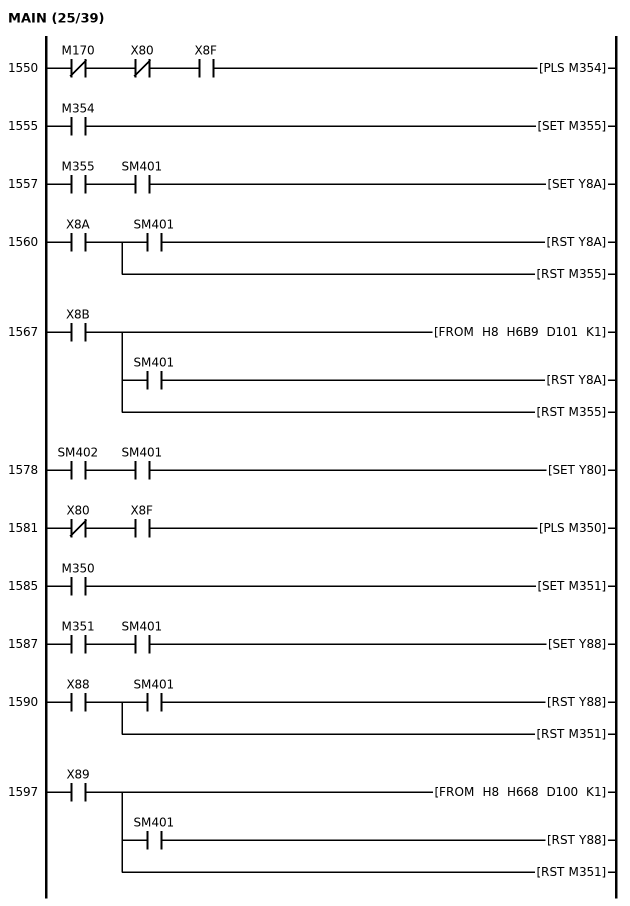
[picture p24: ladder of MAIN, rungs at steps 1550 to 1597]
1550  LDI     M170
      ANI     X80
      AND     X8F
      PLS     M354
1555  LD      M354
      SET     M355
1557  LD      M355
      AND     SM401
      SET     Y8A
1560  LD      X8A
      MPS
      AND     SM401
      RST     Y8A
      MPP
      RST     M355
; 
1567  LD      X8B
      FROM    H8 H6B9 D101 K1
      MPS
      AND     SM401
      RST     Y8A
      MPP
      RST     M355
1578  LD      SM402
      AND     SM401
      SET     Y80
1581  LDI     X80
      AND     X8F
      PLS     M350
1585  LD      M350
      SET     M351
1587  LD      M351
      AND     SM401
      SET     Y88
1590  LD      X88
      MPS
      AND     SM401
      RST     Y88
      MPP
      RST     M351
; 
1597  LD      X89
      FROM    H8 H668 D100 K1
      MPS
      AND     SM401
      RST     Y88
      MPP
      RST     M351
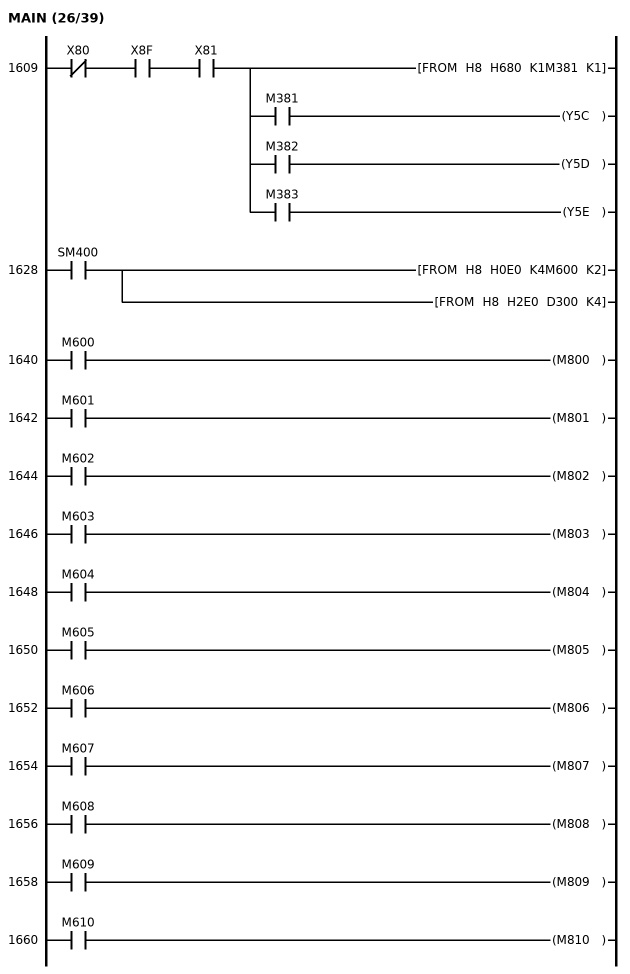
; 
1609  LDI     X80
      AND     X8F
      AND     X81
      FROM    H8 H680 K1M381 K1
      MPS
      AND     M381
      OUT     Y5C
      MRD
      AND     M382
      OUT     Y5D
      MPP
      AND     M383
      OUT     Y5E
; 
1628  LD      SM400
      FROM    H8 H0E0 K4M600 K2
      FROM    H8 H2E0 D300 K4
1640  LD      M600
      OUT     M800
1642  LD      M601
      OUT     M801
1644  LD      M602
      OUT     M802
1646  LD      M603
      OUT     M803
1648  LD      M604
      OUT     M804
1650  LD      M605
      OUT     M805
1652  LD      M606
      OUT     M806
1654  LD      M607
      OUT     M807
1656  LD      M608
      OUT     M808
1658  LD      M609
      OUT     M809
1660  LD      M610
      OUT     M810
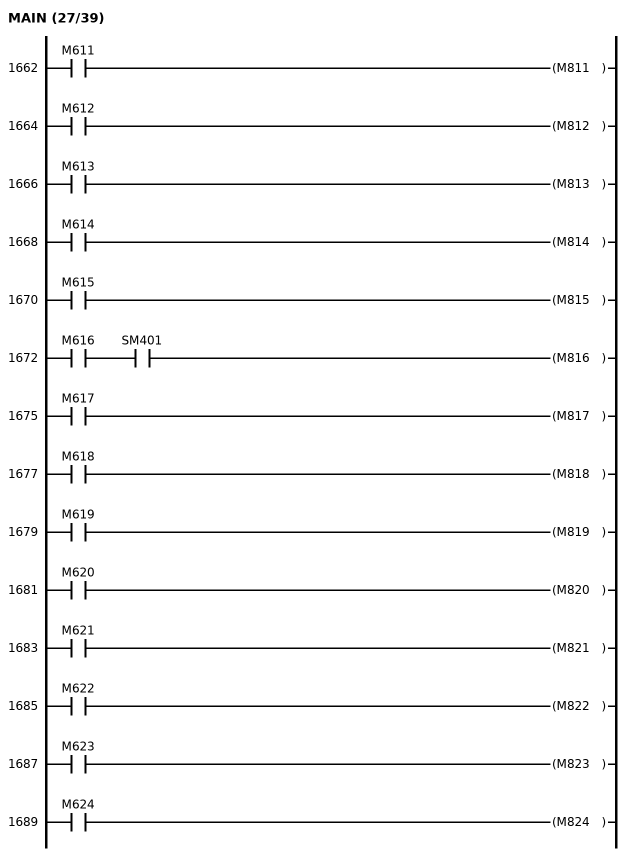
1662  LD      M611
      OUT     M811
1664  LD      M612
      OUT     M812
1666  LD      M613
      OUT     M813
1668  LD      M614
      OUT     M814
1670  LD      M615
      OUT     M815
1672  LD      M616
      AND     SM401
      OUT     M816
1675  LD      M617
      OUT     M817
1677  LD      M618
      OUT     M818
1679  LD      M619
      OUT     M819
1681  LD      M620
      OUT     M820
1683  LD      M621
      OUT     M821
1685  LD      M622
      OUT     M822
1687  LD      M623
      OUT     M823
1689  LD      M624
      OUT     M824
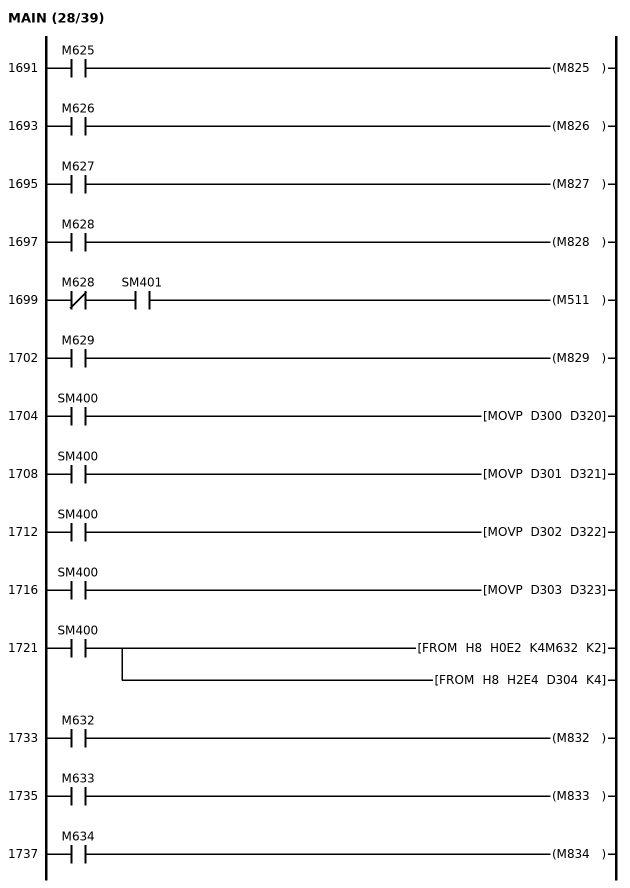
1691  LD      M625
      OUT     M825
1693  LD      M626
      OUT     M826
1695  LD      M627
      OUT     M827
1697  LD      M628
      OUT     M828
1699  LDI     M628
      AND     SM401
      OUT     M511
1702  LD      M629
      OUT     M829
1704  LD      SM400
      MOVP    D300 D320
1708  LD      SM400
      MOVP    D301 D321
1712  LD      SM400
      MOVP    D302 D322
1716  LD      SM400
      MOVP    D303 D323
; 
1721  LD      SM400
      FROM    H8 H0E2 K4M632 K2
      FROM    H8 H2E4 D304 K4
1733  LD      M632
      OUT     M832
1735  LD      M633
      OUT     M833
1737  LD      M634
      OUT     M834
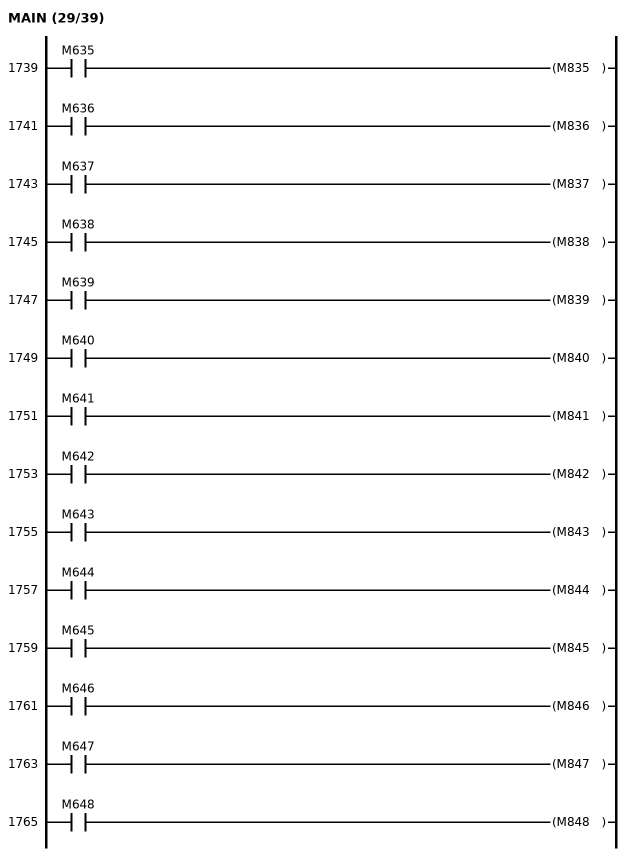
1739  LD      M635
      OUT     M835
1741  LD      M636
      OUT     M836
1743  LD      M637
      OUT     M837
1745  LD      M638
      OUT     M838
1747  LD      M639
      OUT     M839
1749  LD      M640
      OUT     M840
1751  LD      M641
      OUT     M841
1753  LD      M642
      OUT     M842
1755  LD      M643
      OUT     M843
1757  LD      M644
      OUT     M844
1759  LD      M645
      OUT     M845
1761  LD      M646
      OUT     M846
1763  LD      M647
      OUT     M847
1765  LD      M648
      OUT     M848
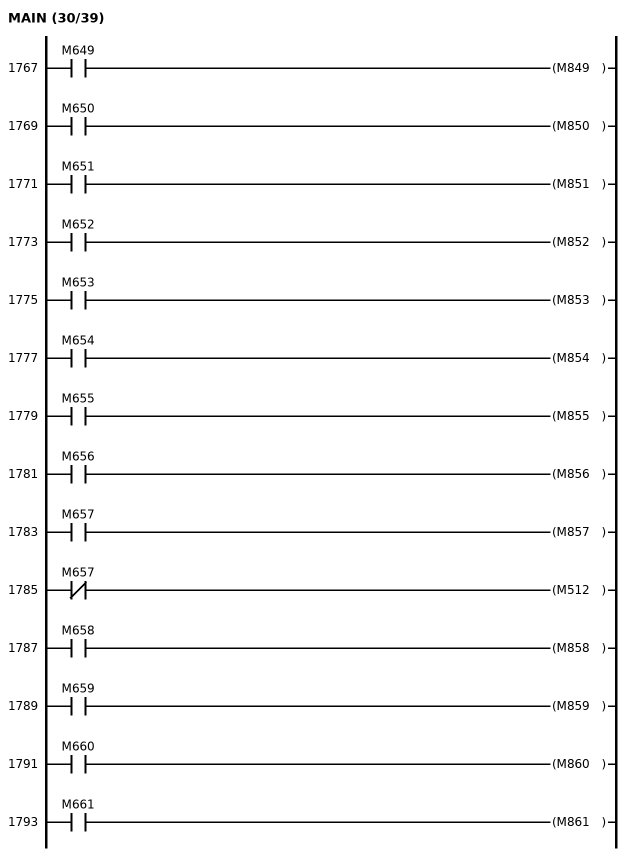
1767  LD      M649
      OUT     M849
1769  LD      M650
      OUT     M850
1771  LD      M651
      OUT     M851
1773  LD      M652
      OUT     M852
1775  LD      M653
      OUT     M853
1777  LD      M654
      OUT     M854
1779  LD      M655
      OUT     M855
1781  LD      M656
      OUT     M856
1783  LD      M657
      OUT     M857
1785  LDI     M657
      OUT     M512
1787  LD      M658
      OUT     M858
1789  LD      M659
      OUT     M859
1791  LD      M660
      OUT     M860
1793  LD      M661
      OUT     M861
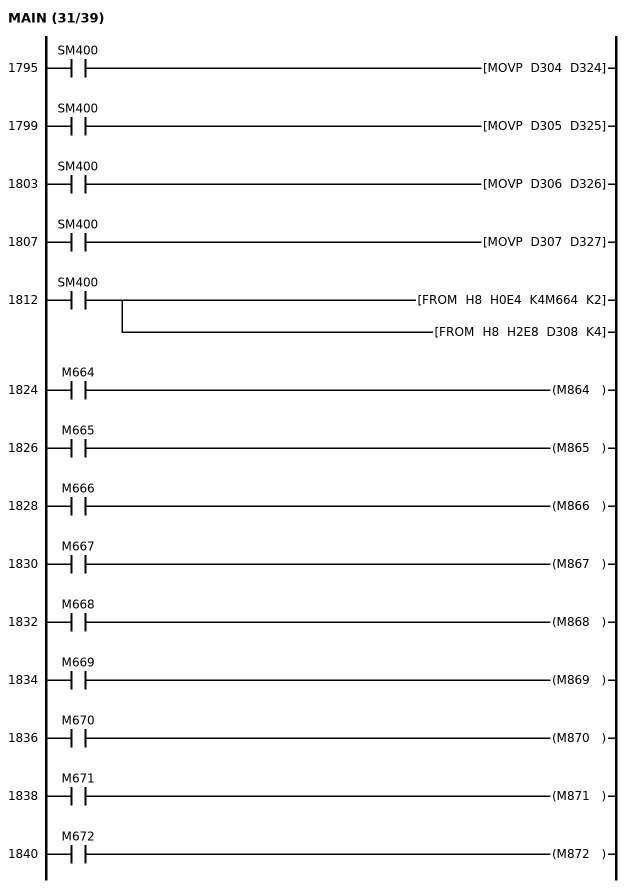
1795  LD      SM400
      MOVP    D304 D324
1799  LD      SM400
      MOVP    D305 D325
1803  LD      SM400
      MOVP    D306 D326
1807  LD      SM400
      MOVP    D307 D327
; 
1812  LD      SM400
      FROM    H8 H0E4 K4M664 K2
      FROM    H8 H2E8 D308 K4
1824  LD      M664
      OUT     M864
1826  LD      M665
      OUT     M865
1828  LD      M666
      OUT     M866
1830  LD      M667
      OUT     M867
1832  LD      M668
      OUT     M868
1834  LD      M669
      OUT     M869
1836  LD      M670
      OUT     M870
1838  LD      M671
      OUT     M871
1840  LD      M672
      OUT     M872
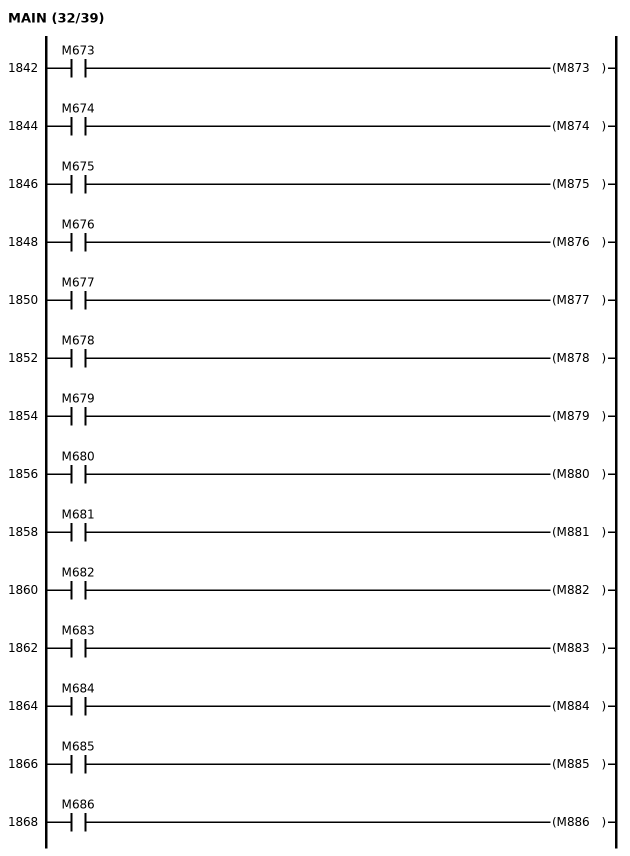
1842  LD      M673
      OUT     M873
1844  LD      M674
      OUT     M874
1846  LD      M675
      OUT     M875
1848  LD      M676
      OUT     M876
1850  LD      M677
      OUT     M877
1852  LD      M678
      OUT     M878
1854  LD      M679
      OUT     M879
1856  LD      M680
      OUT     M880
1858  LD      M681
      OUT     M881
1860  LD      M682
      OUT     M882
1862  LD      M683
      OUT     M883
1864  LD      M684
      OUT     M884
1866  LD      M685
      OUT     M885
1868  LD      M686
      OUT     M886
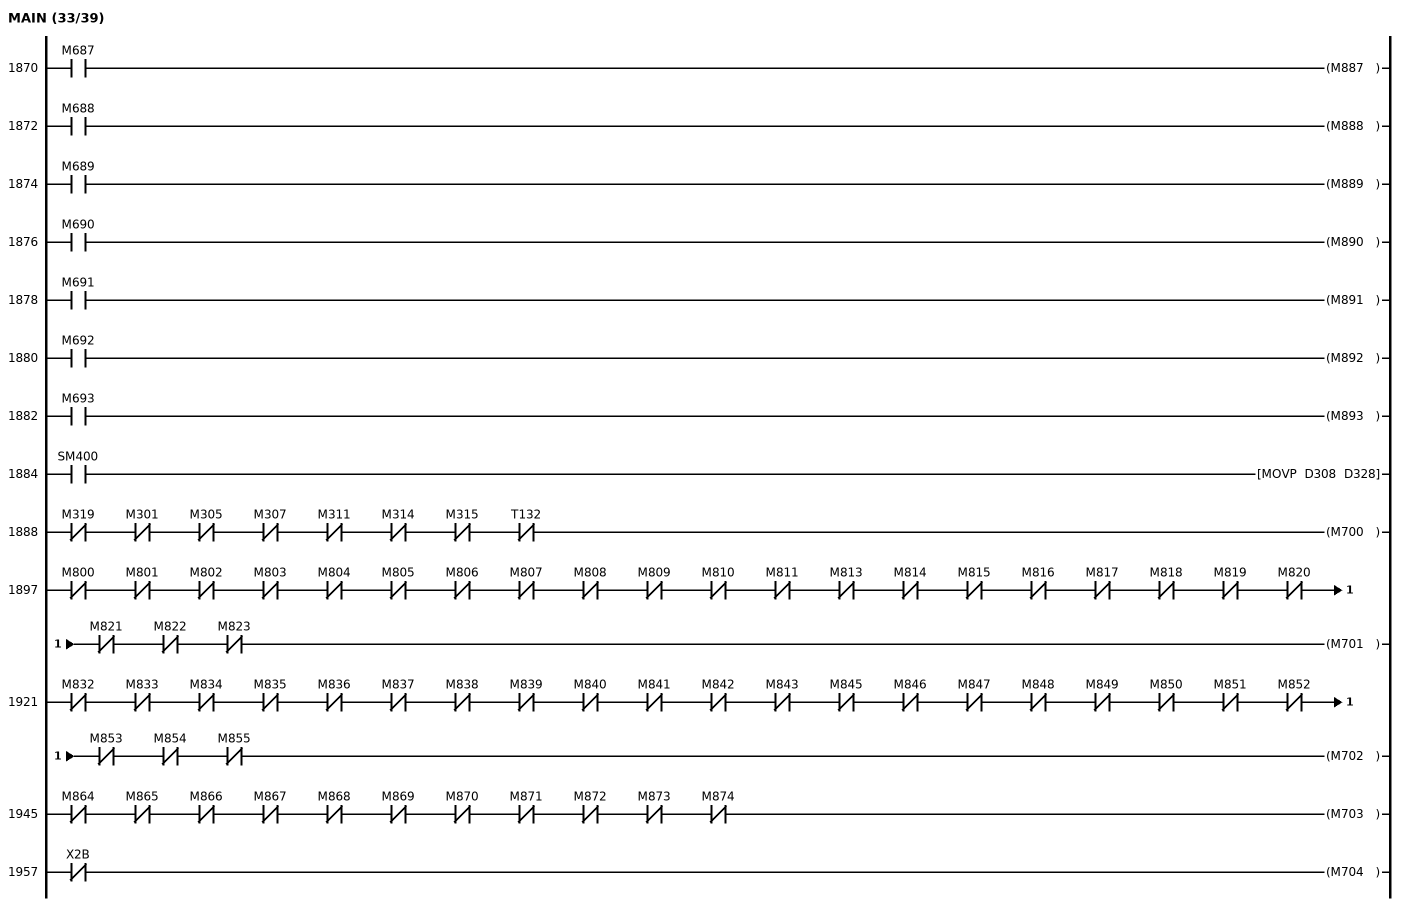
1870  LD      M687
      OUT     M887
1872  LD      M688
      OUT     M888
1874  LD      M689
      OUT     M889
1876  LD      M690
      OUT     M890
1878  LD      M691
      OUT     M891
1880  LD      M692
      OUT     M892
1882  LD      M693
      OUT     M893
1884  LD      SM400
      MOVP    D308 D328
1888  LDI     M319
      ANI     M301
      ANI     M305
      ANI     M307
      ANI     M311
      ANI     M314
      ANI     M315
      ANI     T132
      OUT     M700
1897  LDI     M800
      ANI     M801
      ANI     M802
      ANI     M803
      ANI     M804
      ANI     M805
      ANI     M806
      ANI     M807
      ANI     M808
      ANI     M809
      ANI     M810
      ANI     M811
      ANI     M813
      ANI     M814
      ANI     M815
      ANI     M816
      ANI     M817
      ANI     M818
      ANI     M819
      ANI     M820
      ANI     M821
      ANI     M822
      ANI     M823
      OUT     M701
1921  LDI     M832
      ANI     M833
      ANI     M834
      ANI     M835
      ANI     M836
      ANI     M837
      ANI     M838
      ANI     M839
      ANI     M840
      ANI     M841
      ANI     M842
      ANI     M843
      ANI     M845
      ANI     M846
      ANI     M847
      ANI     M848
      ANI     M849
      ANI     M850
      ANI     M851
      ANI     M852
      ANI     M853
      ANI     M854
      ANI     M855
      OUT     M702
1945  LDI     M864
      ANI     M865
      ANI     M866
      ANI     M867
      ANI     M868
      ANI     M869
      ANI     M870
      ANI     M871
      ANI     M872
      ANI     M873
      ANI     M874
      OUT     M703
1957  LDI     X2B
      OUT     M704
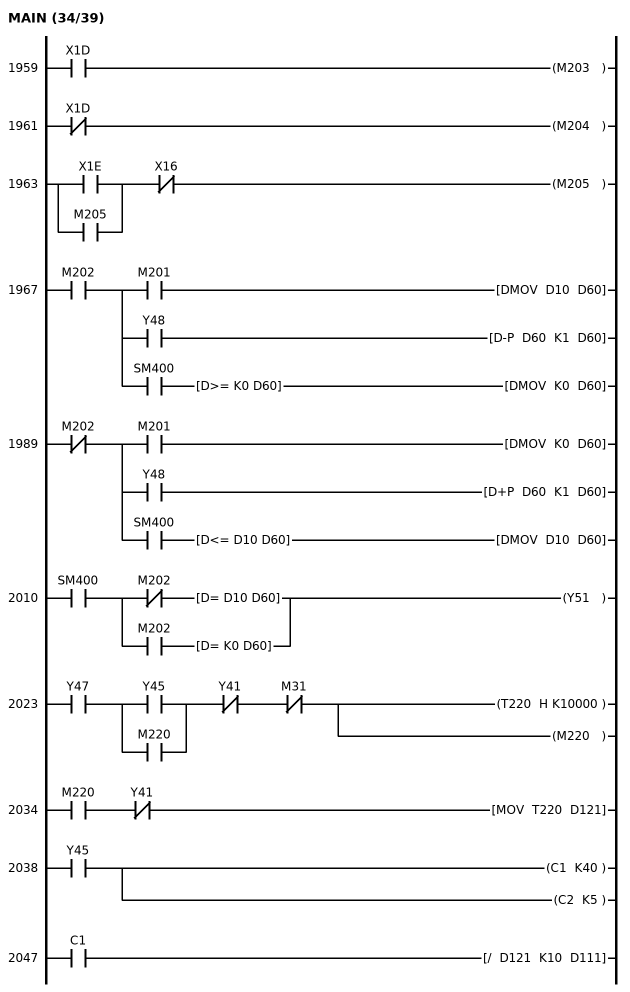
1959  LD      X1D
      OUT     M203
1961  LDI     X1D
      OUT     M204
1963  LD      X1E
      OR      M205
      ANI     X16
      OUT     M205
1967  LD      M202
      MPS
      AND     M201
      DMOV    D10 D60
      MRD
      AND     Y48
      D-P     D60 K1 D60
      MPP
      AND     SM400
      ANDD>=  K0 D60
      DMOV    K0 D60
1989  LDI     M202
      MPS
      AND     M201
      DMOV    K0 D60
      MRD
      AND     Y48
      D+P     D60 K1 D60
      MPP
      AND     SM400
      ANDD<=  D10 D60
      DMOV    D10 D60
2010  LD      SM400
      LDI     M202
      ANDD=   D10 D60
      LD      M202
      ANDD=   K0 D60
      ORB
      ANB
      OUT     Y51
2023  LD      Y47
      LD      Y45
      OR      M220
      ANB
      ANI     Y41
      ANI     M31
      OUTH    T220 K10000
      OUT     M220
2034  LD      M220
      ANI     Y41
      MOV     T220 D121
2038  LD      Y45
      OUT     C1 K40
      OUT     C2 K5
2047  LD      C1
      /       D121 K10 D111
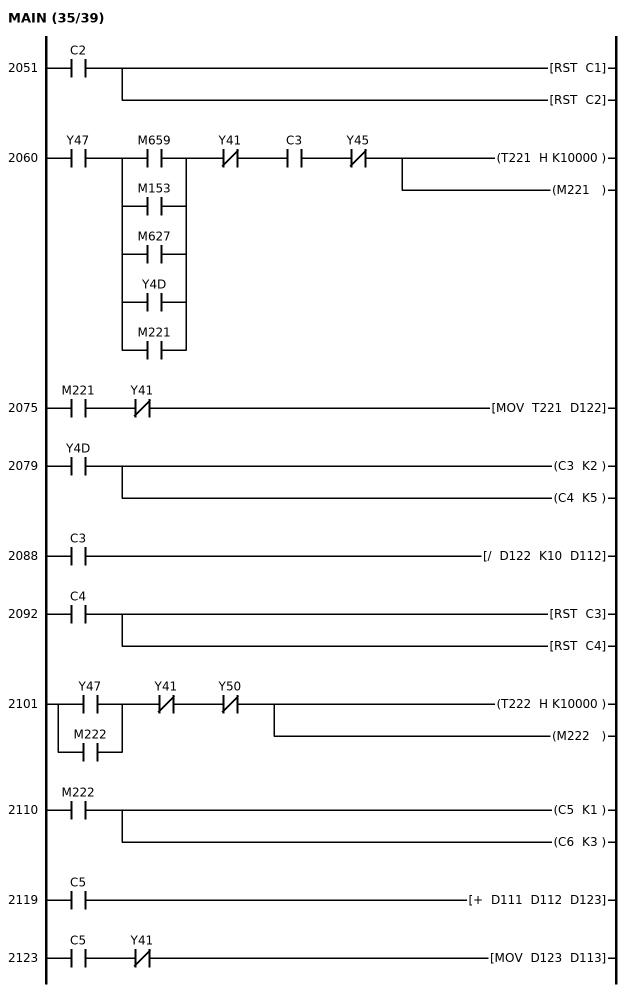
2051  LD      C2
      RST     C1
      RST     C2
2060  LD      Y47
      LD      M659
      OR      M153
      OR      M627
      OR      Y4D
      OR      M221
      ANB
      ANI     Y41
      AND     C3
      ANI     Y45
      OUTH    T221 K10000
      OUT     M221
2075  LD      M221
      ANI     Y41
      MOV     T221 D122
2079  LD      Y4D
      OUT     C3 K2
      OUT     C4 K5
2088  LD      C3
      /       D122 K10 D112
2092  LD      C4
      RST     C3
      RST     C4
2101  LD      Y47
      OR      M222
      ANI     Y41
      ANI     Y50
      OUTH    T222 K10000
      OUT     M222
2110  LD      M222
      OUT     C5 K1
      OUT     C6 K3
2119  LD      C5
      +       D111 D112 D123
2123  LD      C5
      ANI     Y41
      MOV     D123 D113
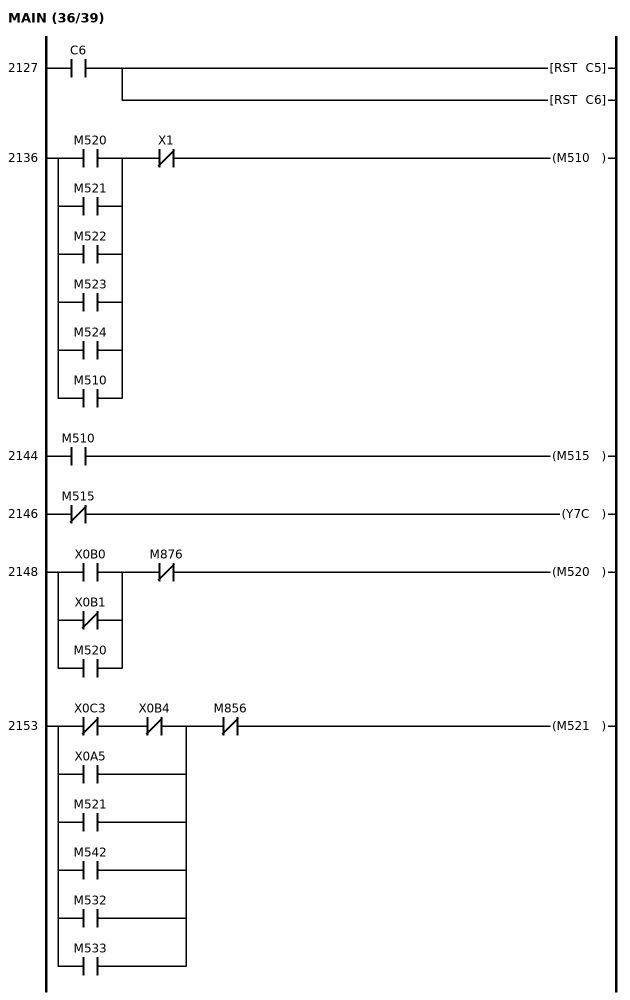
2127  LD      C6
      RST     C5
      RST     C6
2136  LD      M520
      OR      M521
      OR      M522
      OR      M523
      OR      M524
      OR      M510
      ANI     X1
      OUT     M510
2144  LD      M510
      OUT     M515
2146  LDI     M515
      OUT     Y7C
2148  LD      X0B0
      ORI     X0B1
      OR      M520
      ANI     M876
      OUT     M520
2153  LDI     X0C3
      ANI     X0B4
      OR      X0A5
      OR      M521
      OR      M542
      OR      M532
      OR      M533
      ANI     M856
      OUT     M521
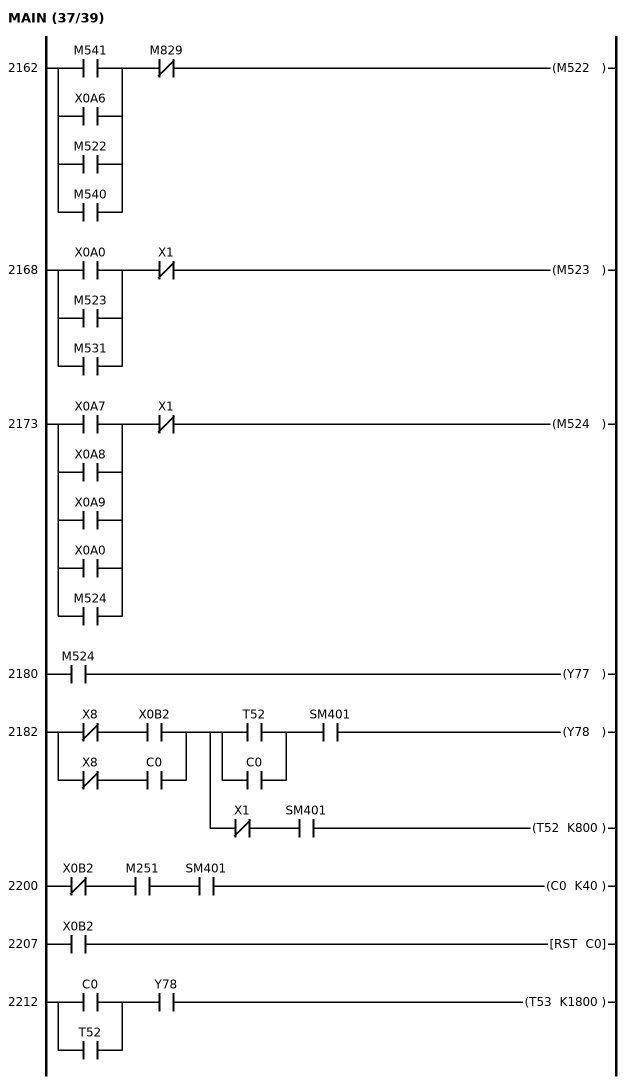
2162  LD      M541
      OR      X0A6
      OR      M522
      OR      M540
      ANI     M829
      OUT     M522
2168  LD      X0A0
      OR      M523
      OR      M531
      ANI     X1
      OUT     M523
2173  LD      X0A7
      OR      X0A8
      OR      X0A9
      OR      X0A0
      OR      M524
      ANI     X1
      OUT     M524
2180  LD      M524
      OUT     Y77
2182  LDI     X8
      AND     X0B2
      LDI     X8
      AND     C0
      ORB
      MPS
      LD      T52
      OR      C0
      ANB
      AND     SM401
      OUT     Y78
      MPP
      ANI     X1
      AND     SM401
      OUT     T52 K800
2200  LDI     X0B2
      AND     M251
      AND     SM401
      OUT     C0 K40
2207  LD      X0B2
      RST     C0
2212  LD      C0
      OR      T52
      AND     Y78
      OUT     T53 K1800
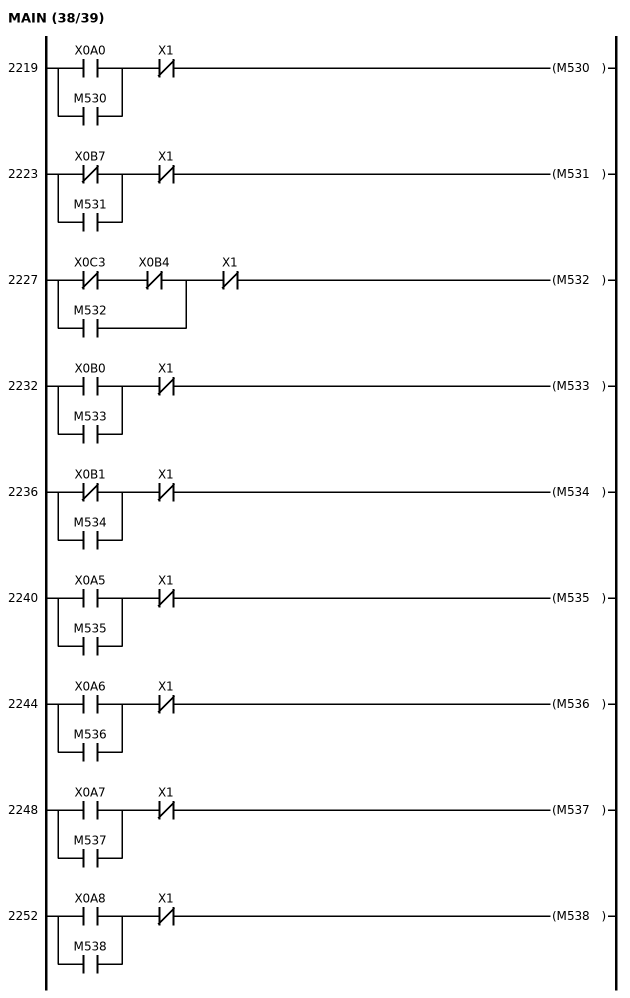
2219  LD      X0A0
      OR      M530
      ANI     X1
      OUT     M530
2223  LDI     X0B7
      OR      M531
      ANI     X1
      OUT     M531
2227  LDI     X0C3
      ANI     X0B4
      OR      M532
      ANI     X1
      OUT     M532
2232  LD      X0B0
      OR      M533
      ANI     X1
      OUT     M533
2236  LDI     X0B1
      OR      M534
      ANI     X1
      OUT     M534
2240  LD      X0A5
      OR      M535
      ANI     X1
      OUT     M535
2244  LD      X0A6
      OR      M536
      ANI     X1
      OUT     M536
2248  LD      X0A7
      OR      M537
      ANI     X1
      OUT     M537
2252  LD      X0A8
      OR      M538
      ANI     X1
      OUT     M538
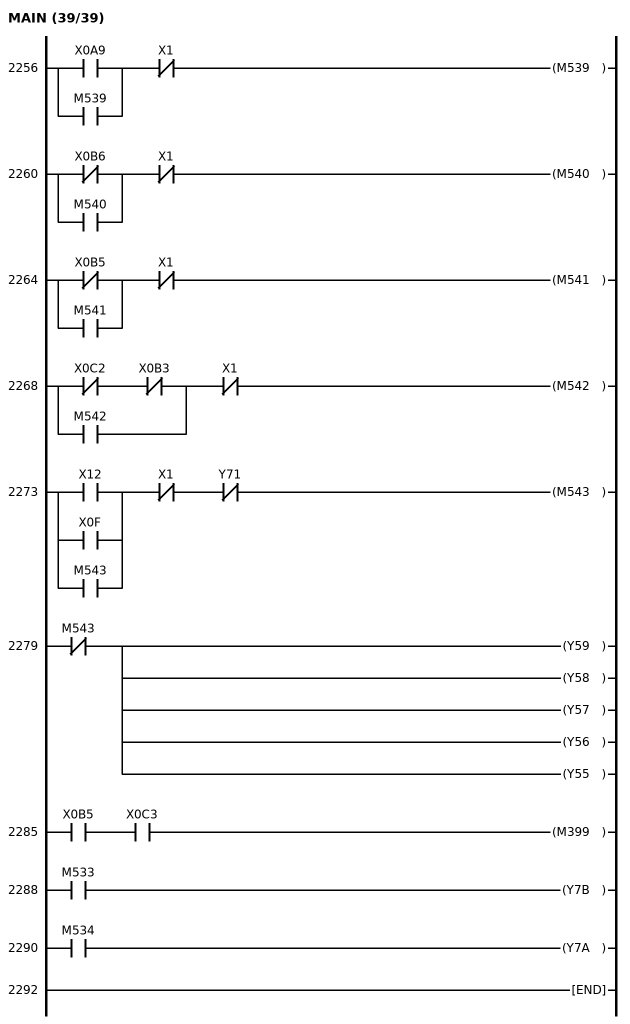
2256  LD      X0A9
      OR      M539
      ANI     X1
      OUT     M539
2260  LDI     X0B6
      OR      M540
      ANI     X1
      OUT     M540
2264  LDI     X0B5
      OR      M541
      ANI     X1
      OUT     M541
2268  LDI     X0C2
      ANI     X0B3
      OR      M542
      ANI     X1
      OUT     M542
2273  LD      X12
      OR      X0F
      OR      M543
      ANI     X1
      ANI     Y71
      OUT     M543
2279  LDI     M543
      OUT     Y59
      OUT     Y58
      OUT     Y57
      OUT     Y56
      OUT     Y55
2285  LD      X0B5
      AND     X0C3
      OUT     M399
2288  LD      M533
      OUT     Y7B
2290  LD      M534
      OUT     Y7A
2292  END
END_PROGRAM
